// TwinCAT 3 PLC project PLC_PML
// ProgramVersion: 3.1.4023.0
// libraries:
//   PML_Base_Library, * (SPT)
//   Tc2_Math, * (Beckhoff Automation GmbH)
//   Tc2_MC2, * (Beckhoff Automation GmbH)
//   Tc2_MC2_Drive, * (Beckhoff Automation GmbH)
//   Tc2_Standard, * (Beckhoff Automation GmbH)
//   Tc2_System, * (Beckhoff Automation GmbH)
//   Tc2_Utilities, * (Beckhoff Automation GmbH)
//   Tc3_EventLogger, * (Beckhoff Automation GmbH)
//   Tc3_Module, * (Beckhoff Automation GmbH)
//   Tc3_PackML_V2, * (Beckhoff Automation GmbH)
// project tree:
//   Application/01_Application_Level_Items/02_DUT/01_ENUM/ E_PMLUnitMode.TcDUT (not stored)
//   Application/01_Application_Level_Items/02_DUT/02_STRUCT/ ST_ProductionData_HMI.TcDUT
//   Application/01_Application_Level_Items/02_DUT/03_ALIAS/ T_PackMLTags.TcDUT (not stored)
//   Application/01_Application_Level_Items/03_ITFs/ ITF_ProductionData.TcIO
//   Application/01_Application_Level_Items/04_HMI_Connections/ FB_MainModule_HMI_Connection.TcPOU (not stored), ST_PMLControl.TcDUT, ST_PMLControl_Simplified.TcDUT
//   Application/01_Application_Level_Items/999_VISU/ V_Application.TcVIS (not stored)
//   Application/01_Application_Level_Items/99_Templates/ FB_Module_TEMPLATE.TcPOU
//   Application/01_Application_Level_Items/ FB_ProductionMonitor.TcPOU
//   Application/02_MachineModules/ FB_TestMachine.TcPOU (not stored)
//   Application/03_EquipmentModules/ FB_TestEquipment.TcPOU (not stored)
//   Application/04_Components/01_Cylinder_Example/ FB_CylinderBase.TcPOU (not stored), ITF_CylinderBase.TcIO (not stored), ST_CylinderBase_HMI.TcDUT (not stored)
//   Application/ MAIN.TcPOU (not stored)
//   / GlobalTextList.TcGTLO (not stored), PlcTask.TcTTO (not stored), Visualization Manager.TcVMO (not stored)
// real-time tasks:
//   TASK PlcTask: cycle T#1ms, priority 20, ADS port 350
//   TASK VISU_TASK: cycle T#200000us, priority 30, ADS port 351
//   TASK Job Task: cycle default, priority 32
//   TASK MC-Task (MET): cycle T#2ms, priority 3, ADS port 521
//   TASK MC-Task (MPT): cycle T#10ms, priority 8, ADS port 531
// motion (NC):
//   TASK NC-Task 1 SAF: cycle T#2ms, priority 4, ADS port 501
//   TASK NC-Task 1 SVB: cycle T#10ms, priority 9, ADS port 511
//   AXIS Axis 1 (id 1)
//     General: UnitFlags=#x00000004
//     Dynamic: AccelerationMaximum=10000, DecelerationMaximum=10000, Acceleration=1000, Deceleration=1000, Jerk=1750
//     Velo: Maximum=1500
//     OtherSettings: AllowMotionCmdToSlave=true
//     encoder EncType=1
//       EncPara: ModuloFactor=720
//     drive DrvType=5
//       Analog: TorqueSetpointScale=10, ScaleFactorActTorque=0.1
//       TimeComp: TaskDelayCycles=1
//     controller CtrType=1
//       CtrPara: PriorControlFactor=1
//         Observer: BandWidth=20
//   AXIS Axis 2 (id 2)
//     General: UnitFlags=#x00000004
//     OtherSettings: AllowMotionCmdToSlave=true
//     encoder EncType=1
//     drive DrvType=5
//       Analog: TorqueSetpointScale=10, ScaleFactorActTorque=0.1
//       TimeComp: TaskDelayCycles=1
//     controller CtrType=1
//       CtrPara: PriorControlFactor=1
//         Observer: BandWidth=20

// ---- Application/01_Application_Level_Items/02_DUT/02_STRUCT/ST_ProductionData_HMI.TcDUT
TYPE ST_ProductionData_HMI :
    STRUCT
        bHMIControlAvailable    : BOOL; //Set TRUE *FROM PLC* when HMI requests can be processed
        bIncomingHMIRequest     : BOOL; //Pulses TRUE when an HMI request is issued
        bHMICommandConfirmation : BOOL; //Confirms receipt and subsequent processing of the command sent by the HMI

        bShiftLengthHMISetRequest : BOOL;
        tShiftLengthHMISetValue   : TIME;

        bShiftProductionTargetHMISetRequest : BOOL;
        nShiftProductionTargetHMISetValue   : DINT;

        bWarningMarginHMISetRequest : BOOL;
        fWarningMarginHMISetValue   : LREAL;

        bProductionRateHMISetRequest : BOOL;
        fProductionRateHMISetValue   : LREAL;

        tShiftLength           : TIME; //Specify the time duration of a shift
        nShiftProductionTarget : DINT; //Specify the desired production count by end of shift

        nCurrentAcceptableProductionCount : DINT;
        nCurrentWarningProductionCount    : DINT;
        nCurrentShiftProductionCount      : DINT; //Number of products completed so far on the current shift
        nCurrentShiftTarget               : DINT; //Expected number of completed products at the current time in the shift
        tCurrentShiftTime                 : TIME; //Time elapsed since the start of the shift
        tRemainingShiftTime               : TIME; //Time remaining in the current shift
        tShiftStartTimeStamp              : TIMESTRUCT;
        tShiftStartTimeStamp_UTC          : STRING;
        fProductionRate_Setpoint          : LREAL;
        fProductionRate_Actual            : LREAL;
        fProductionRate_Required          : LREAL;

    END_STRUCT
END_TYPE

// ---- Application/01_Application_Level_Items/04_HMI_Connections/ST_PMLControl.TcDUT
TYPE ST_PMLControl :
    STRUCT
        bNewCommand   : BOOL;
        bConfirmation : BOOL;

        eMode        : E_PMLUnitMode;
        eModeCommand : E_PMLUnitMode;

        eState        : E_PMLState;
        eStateCommand : E_PMLCommand;

        a_sModeNames : ARRAY[0..31] OF STRING;
    END_STRUCT
END_TYPE

// ---- Application/01_Application_Level_Items/04_HMI_Connections/ST_PMLControl_Simplified.TcDUT
TYPE ST_PMLControl_Simplified :
    STRUCT
        bConfirmation : BOOL;

        bClearEnabled : BOOL;
        bResetEnabled : BOOL;
        bStartEnabled : BOOL;
        bStopEnabled  : BOOL;

        bClearPressed : BOOL;
        bResetPressed : BOOL;
        bStartPressed : BOOL;
        bStopPressed  : BOOL;
    END_STRUCT
END_TYPE

// ---- Application/01_Application_Level_Items/03_ITFs/ITF_ProductionData.TcIO
INTERFACE ITF_ProductionData

PROPERTY CurrentShiftAcceptableProduction : DINT
GET
END_GET
SET
END_SET
END_PROPERTY

PROPERTY CurrentShiftProductionCount : DINT
GET
END_GET
END_PROPERTY

PROPERTY CurrentShiftTarget : DINT
GET
END_GET
END_PROPERTY

PROPERTY CurrentShiftTime : TIME
GET
END_GET
END_PROPERTY

PROPERTY CurrentShiftWarningProduction : DINT
GET
END_GET
SET
END_SET
END_PROPERTY

PROPERTY NewProductionRate : bool
GET
END_GET
END_PROPERTY

PROPERTY ProductComplete : bool
GET
END_GET
SET
END_SET
END_PROPERTY

PROPERTY ProductionRate_Actual : lreal
GET
END_GET
END_PROPERTY

PROPERTY ProductionRate_Required : lreal
GET
END_GET
SET
END_SET
END_PROPERTY

PROPERTY ProductionRate_Setpoint : lreal
GET
END_GET
SET
END_SET
END_PROPERTY

PROPERTY RateAveragingCount : DINT
GET
END_GET
SET
END_SET
END_PROPERTY

PROPERTY RemainingShiftTime : TIME
GET
END_GET
SET
END_SET
END_PROPERTY

PROPERTY ShiftComplete : BOOL
GET
END_GET
END_PROPERTY

PROPERTY ShiftLength : TIME
GET
END_GET
SET
END_SET
END_PROPERTY

PROPERTY ShiftProductionTarget : DINT
GET
END_GET
SET
END_SET
END_PROPERTY

PROPERTY WarningMargin : LREAL //0 to 100, interpreted as a percentage difference between the current rate and the required rate to meet the production target, decimal values permitted
GET
END_GET
SET
END_SET
END_PROPERTY

END_INTERFACE

// ---- Application/01_Application_Level_Items/99_Templates/FB_Module_TEMPLATE.TcPOU
FUNCTION_BLOCK FB_Module_TEMPLATE EXTENDS FB_PMLModuleBase
VAR
    //Define the Sub modules here for this module. (If any)  Also set the Interfaces in the initialize method.
    (*fbSubModule1				: FB_ApplicationModule_TEMPLATE := (ModuleName :=  'Test Module 1');
	*)
    (*fbSubModule2				: FB_ApplicationModule_TEMPLATE := (ModuleName :=  'Test Module 2');
	*)
    //temporary array of module base interfaces to be copied over to the base class a_itfPackMLBase variable
    a_ITF_PackMLBase_init : ARRAY[1..MAX_NO_OF_SUBMODULES] OF ITF_PMLModuleBase
        := [ (*	fbSubModule1,
																							 	fbSubModule2*) ];

    //Define the components here for this module. (If any) Also set the Interfaces in the initialize method.
    (*fbComponent1				: FB_ComponentBase (Extension):= (Name := 'Test Component 1');
	*)
    (*fbComponent2				: FB_ComponentBase (Extension):= (Name := 'Test Component 2');
	*)
    //temporary array of module base interfaces to be copied over to the base class a_itfPackMLBase variable
    a_ITF_Components_init : ARRAY[1..GVL_PML_Base.MAX_NO_OF_COMPONENTS] OF ITF_ComponentBase := [ (*	fbComponent1,
																											fbComponent2*)
    ];

END_VAR

//*********************************************************
//Body of block is not called by base code, only implement application
//code in CyclicUpdate or in methods called by it or its subcalls
//*********************************************************

METHOD Aborted
CASE eMode OF
    //	====================================================================PRODUCTION MODE=========================================================	
    E_PMLUnitMode.ePMLUnitMode_Production:
        ;
    //	====================================================================MANUAL MODE=============================================================	
    E_PMLUnitMode.ePMLUnitMode_Manual:
        ;
    //	=====================================================================MAINTENANCE MODE=======================================================	
    E_PMLUnitMode.ePMLUnitMode_Maintenance:
        ;
    //	=====================================================================CUSTOM MODE 1==========================================================	
    (*	E_PMLUnitMode.ePMLUnitMode_YOURCUSTOMMODE		
		;*)
    //	======================================================================INVALID MODE==========================================================	
    E_PMLUnitMode.ePMLUnitMode_Invalid:
        ;
END_CASE
END_METHOD

METHOD Aborting
//bNoStateTasksToComplete := TRUE;		// Change to False if not used

//Implement state Tasks here
(*
IF (insert your completion conditions) THEN

bStateTasksComplete := TRUE;				//Once these actions are completed successfully, set bStateTasksComplete to allow the base code to advance once all children have also reached the proper state

END_IF
*)

SUPER^.Aborting();

(*	Reference State Machine for mode specific actions - Be sure to paste above the SUPER^ Call if used - Delete if not needed

CASE eMode OF
//	====================================================================PRODUCTION MODE=========================================================	
	E_PMLUnitMode.ePMLUnitMode_Production:			
		;
//	====================================================================MANUAL MODE=============================================================	
	E_PMLUnitMode.ePMLUnitMode_Manual:				
		;
//	=====================================================================MAINTENANCE MODE=======================================================	
	E_PMLUnitMode.ePMLUnitMode_Maintenance:			
		;	
//	=====================================================================CUSTOM MODE 1==========================================================	
(*	E_PMLUnitMode.ePMLUnitMode_YOURCUSTOMMODE		
		;*)
//	======================================================================INVALID MODE==========================================================	
	E_PMLUnitMode.ePMLUnitMode_Invalid:				
		;
END_CASE
*)
END_METHOD

METHOD Clearing
//bNoStateTasksToComplete := TRUE;		// Change to False if not used

//Implement state Tasks here
(*
IF (insert your completion conditions) THEN

bStateTasksComplete := TRUE;				//Once these actions are completed successfully, set bStateTasksComplete to allow the base code to advance once all children have also reached the proper state

END_IF
*)

SUPER^.Clearing();
(*	Reference State Machine for mode specific actions - Be sure to paste above the SUPER^ Call if used - Delete if not needed

CASE eMode OF
//	====================================================================PRODUCTION MODE=========================================================	
	E_PMLUnitMode.ePMLUnitMode_Production:			
		;
//	====================================================================MANUAL MODE=============================================================	
	E_PMLUnitMode.ePMLUnitMode_Manual:				
		;
//	=====================================================================MAINTENANCE MODE=======================================================	
	E_PMLUnitMode.ePMLUnitMode_Maintenance:			
		;	
//	=====================================================================CUSTOM MODE 1==========================================================	
(*	E_PMLUnitMode.ePMLUnitMode_YOURCUSTOMMODE		
		;*)
//	======================================================================INVALID MODE==========================================================	
	E_PMLUnitMode.ePMLUnitMode_Invalid:				
		;
END_CASE
*)
END_METHOD

METHOD Complete
CASE eMode OF
    //	====================================================================PRODUCTION MODE=========================================================	
    E_PMLUnitMode.ePMLUnitMode_Production:
        ;
    //	====================================================================MANUAL MODE=============================================================	
    E_PMLUnitMode.ePMLUnitMode_Manual:
        ;
    //	=====================================================================MAINTENANCE MODE=======================================================	
    E_PMLUnitMode.ePMLUnitMode_Maintenance:
        ;
    //	=====================================================================CUSTOM MODE 1==========================================================	
    (*	E_PMLUnitMode.ePMLUnitMode_YOURCUSTOMMODE		
		;*)
    //	======================================================================INVALID MODE==========================================================	
    E_PMLUnitMode.ePMLUnitMode_Invalid:
        ;
END_CASE
END_METHOD

METHOD Completing
//bNoStateTasksToComplete := TRUE;		// Change to False if not used

//Implement state Tasks here
(*
IF (insert your completion conditions) THEN

bStateTasksComplete := TRUE;				//Once these actions are completed successfully, set bStateTasksComplete to allow the base code to advance once all children have also reached the proper state

END_IF
*)

SUPER^.Completing();

(*	Reference State Machine for mode specific actions - Be sure to paste above the SUPER^ Call if used - Delete if not needed

CASE eMode OF
//	====================================================================PRODUCTION MODE=========================================================	
	E_PMLUnitMode.ePMLUnitMode_Production:			
		;
//	====================================================================MANUAL MODE=============================================================	
	E_PMLUnitMode.ePMLUnitMode_Manual:				
		;
//	=====================================================================MAINTENANCE MODE=======================================================	
	E_PMLUnitMode.ePMLUnitMode_Maintenance:			
		;	
//	=====================================================================CUSTOM MODE 1==========================================================	
(*	E_PMLUnitMode.ePMLUnitMode_YOURCUSTOMMODE		
		;*)
//	======================================================================INVALID MODE==========================================================	
	E_PMLUnitMode.ePMLUnitMode_Invalid:				
		;
END_CASE
*)
END_METHOD

// 
// Cyclic Code
METHOD CyclicLogic
VAR
    i : UDINT; //Generic iteration value
END_VAR
// Main loop of the parent module
SUPER^.CyclicLogic();
END_METHOD

METHOD Execute
CASE eMode OF
    //	====================================================================PRODUCTION MODE=========================================================	
    E_PMLUnitMode.ePMLUnitMode_Production:
        ;
    //	====================================================================MANUAL MODE=============================================================	
    E_PMLUnitMode.ePMLUnitMode_Manual:
        ;
    //	=====================================================================MAINTENANCE MODE=======================================================	
    E_PMLUnitMode.ePMLUnitMode_Maintenance:
        ;
    //	=====================================================================CUSTOM MODE 1==========================================================	
    (*	E_PMLUnitMode.ePMLUnitMode_YOURCUSTOMMODE		
		;*)
    //	======================================================================INVALID MODE==========================================================	
    E_PMLUnitMode.ePMLUnitMode_Invalid:
        ;
END_CASE
END_METHOD

METHOD Held
CASE eMode OF
    //	====================================================================PRODUCTION MODE=========================================================	
    E_PMLUnitMode.ePMLUnitMode_Production:
        ;
    //	====================================================================MANUAL MODE=============================================================	
    E_PMLUnitMode.ePMLUnitMode_Manual:
        ;
    //	=====================================================================MAINTENANCE MODE=======================================================	
    E_PMLUnitMode.ePMLUnitMode_Maintenance:
        ;
    //	=====================================================================CUSTOM MODE 1==========================================================	
    (*	E_PMLUnitMode.ePMLUnitMode_YOURCUSTOMMODE		
		;*)
    //	======================================================================INVALID MODE==========================================================	
    E_PMLUnitMode.ePMLUnitMode_Invalid:
        ;
END_CASE
END_METHOD

METHOD Holding
//bNoStateTasksToComplete := TRUE;		// Change to False if not used

//Implement state Tasks here
(*
IF (insert your completion conditions) THEN

bStateTasksComplete := TRUE;				//Once these actions are completed successfully, set bStateTasksComplete to allow the base code to advance once all children have also reached the proper state

END_IF
*)

SUPER^.Holding();

(*	Reference State Machine for mode specific actions - Be sure to paste above the SUPER^ Call if used - Delete if not needed

CASE eMode OF
//	====================================================================PRODUCTION MODE=========================================================	
	E_PMLUnitMode.ePMLUnitMode_Production:			
		;
//	====================================================================MANUAL MODE=============================================================	
	E_PMLUnitMode.ePMLUnitMode_Manual:				
		;
//	=====================================================================MAINTENANCE MODE=======================================================	
	E_PMLUnitMode.ePMLUnitMode_Maintenance:			
		;	
//	=====================================================================CUSTOM MODE 1==========================================================	
(*	E_PMLUnitMode.ePMLUnitMode_YOURCUSTOMMODE		
		;*)
//	======================================================================INVALID MODE==========================================================	
	E_PMLUnitMode.ePMLUnitMode_Invalid:				
		;
END_CASE
*)
END_METHOD

METHOD Idle
CASE eMode OF
    //	====================================================================PRODUCTION MODE=========================================================	
    E_PMLUnitMode.ePMLUnitMode_Production:
        ;
    //	====================================================================MANUAL MODE=============================================================	
    E_PMLUnitMode.ePMLUnitMode_Manual:
        ;
    //	=====================================================================MAINTENANCE MODE=======================================================	
    E_PMLUnitMode.ePMLUnitMode_Maintenance:
        ;
    //	=====================================================================CUSTOM MODE 1==========================================================	
    (*	E_PMLUnitMode.ePMLUnitMode_YOURCUSTOMMODE		
		;*)
    //	======================================================================INVALID MODE==========================================================	
    E_PMLUnitMode.ePMLUnitMode_Invalid:
        ;
END_CASE
END_METHOD

METHOD Initialize
VAR
    i : UDINT; //Generic iteration value
END_VAR
// Define the interfaces to the different subunits (Must take place before SUPER^.initialize call)
FOR i := 1 TO MAX_NO_OF_SUBMODULES DO
    a_ITF_PackMLBase[i] := a_ITF_PackMLBase_init[i];
END_FOR

FOR i := 1 TO MAX_NO_OF_COMPONENTS DO
    a_ITF_Components[i] := a_ITF_Components_init[i];
END_FOR

// Init of the parent class object (Must be called AFTER most local init code, since the sub module interface array assignments should be made here, and then operated on within the module base init
SUPER^.Initialize();
END_METHOD

METHOD Resetting
//bNoStateTasksToComplete := TRUE;		// Change to False if not used

//Implement state Tasks here
(*
IF (insert your completion conditions) THEN

bStateTasksComplete := TRUE;				//Once these actions are completed successfully, set bStateTasksComplete to allow the base code to advance once all children have also reached the proper state

END_IF
*)

SUPER^.Resetting();

(*	Reference State Machine for mode specific actions - Be sure to paste above the SUPER^ Call if used - Delete if not needed

CASE eMode OF
//	====================================================================PRODUCTION MODE=========================================================	
	E_PMLUnitMode.ePMLUnitMode_Production:			
		;
//	====================================================================MANUAL MODE=============================================================	
	E_PMLUnitMode.ePMLUnitMode_Manual:				
		;
//	=====================================================================MAINTENANCE MODE=======================================================	
	E_PMLUnitMode.ePMLUnitMode_Maintenance:			
		;	
//	=====================================================================CUSTOM MODE 1==========================================================	
(*	E_PMLUnitMode.ePMLUnitMode_YOURCUSTOMMODE		
		;*)
//	======================================================================INVALID MODE==========================================================	
	E_PMLUnitMode.ePMLUnitMode_Invalid:				
		;
END_CASE
*)
END_METHOD

METHOD Starting
//bNoStateTasksToComplete := TRUE;		// Change to False if not used

//Implement state Tasks here
(*
IF (insert your completion conditions) THEN

bStateTasksComplete := TRUE;				//Once these actions are completed successfully, set bStateTasksComplete to allow the base code to advance once all children have also reached the proper state

END_IF
*)

SUPER^.Starting();

(*	Reference State Machine for mode specific actions - Be sure to paste above the SUPER^ Call if used - Delete if not needed

CASE eMode OF
//	====================================================================PRODUCTION MODE=========================================================	
	E_PMLUnitMode.ePMLUnitMode_Production:			
		;
//	====================================================================MANUAL MODE=============================================================	
	E_PMLUnitMode.ePMLUnitMode_Manual:				
		;
//	=====================================================================MAINTENANCE MODE=======================================================	
	E_PMLUnitMode.ePMLUnitMode_Maintenance:			
		;	
//	=====================================================================CUSTOM MODE 1==========================================================	
(*	E_PMLUnitMode.ePMLUnitMode_YOURCUSTOMMODE		
		;*)
//	======================================================================INVALID MODE==========================================================	
	E_PMLUnitMode.ePMLUnitMode_Invalid:				
		;
END_CASE
*)
END_METHOD

METHOD Stopped
CASE eMode OF
    //	====================================================================PRODUCTION MODE=========================================================	
    E_PMLUnitMode.ePMLUnitMode_Production:
        ;
    //	====================================================================MANUAL MODE=============================================================	
    E_PMLUnitMode.ePMLUnitMode_Manual:
        ;
    //	=====================================================================MAINTENANCE MODE=======================================================	
    E_PMLUnitMode.ePMLUnitMode_Maintenance:
        ;
    //	=====================================================================CUSTOM MODE 1==========================================================	
    (*	E_PMLUnitMode.ePMLUnitMode_YOURCUSTOMMODE		
		;*)
    //	======================================================================INVALID MODE==========================================================	
    E_PMLUnitMode.ePMLUnitMode_Invalid:
        ;
END_CASE
END_METHOD

METHOD Stopping
//bNoStateTasksToComplete := TRUE;		// Change to False if not used

//Implement state Tasks here
(*
IF (insert your completion conditions) THEN

bStateTasksComplete := TRUE;				//Once these actions are completed successfully, set bStateTasksComplete to allow the base code to advance once all children have also reached the proper state

END_IF
*)

SUPER^.Stopping();

(*	Reference State Machine for mode specific actions - Be sure to paste above the SUPER^ Call if used - Delete if not needed

CASE eMode OF
//	====================================================================PRODUCTION MODE=========================================================	
	E_PMLUnitMode.ePMLUnitMode_Production:			
		;
//	====================================================================MANUAL MODE=============================================================	
	E_PMLUnitMode.ePMLUnitMode_Manual:				
		;
//	=====================================================================MAINTENANCE MODE=======================================================	
	E_PMLUnitMode.ePMLUnitMode_Maintenance:			
		;	
//	=====================================================================CUSTOM MODE 1==========================================================	
(*	E_PMLUnitMode.ePMLUnitMode_YOURCUSTOMMODE		
		;*)
//	======================================================================INVALID MODE==========================================================	
	E_PMLUnitMode.ePMLUnitMode_Invalid:				
		;
END_CASE
*)
END_METHOD

METHOD Suspended
CASE eMode OF
    //	====================================================================PRODUCTION MODE=========================================================	
    E_PMLUnitMode.ePMLUnitMode_Production:
        ;
    //	====================================================================MANUAL MODE=============================================================	
    E_PMLUnitMode.ePMLUnitMode_Manual:
        ;
    //	=====================================================================MAINTENANCE MODE=======================================================	
    E_PMLUnitMode.ePMLUnitMode_Maintenance:
        ;
    //	=====================================================================CUSTOM MODE 1==========================================================	
    (*	E_PMLUnitMode.ePMLUnitMode_YOURCUSTOMMODE		
		;*)
    //	======================================================================INVALID MODE==========================================================	
    E_PMLUnitMode.ePMLUnitMode_Invalid:
        ;
END_CASE
END_METHOD

METHOD Suspending
//bNoStateTasksToComplete := TRUE;		// Change to False if not used

//Implement state Tasks here
(*
IF (insert your completion conditions) THEN

bStateTasksComplete := TRUE;				//Once these actions are completed successfully, set bStateTasksComplete to allow the base code to advance once all children have also reached the proper state

END_IF
*)

SUPER^.Suspending();

(*	Reference State Machine for mode specific actions - Be sure to paste above the SUPER^ Call if used - Delete if not needed

CASE eMode OF
//	====================================================================PRODUCTION MODE=========================================================	
	E_PMLUnitMode.ePMLUnitMode_Production:			
		;
//	====================================================================MANUAL MODE=============================================================	
	E_PMLUnitMode.ePMLUnitMode_Manual:				
		;
//	=====================================================================MAINTENANCE MODE=======================================================	
	E_PMLUnitMode.ePMLUnitMode_Maintenance:			
		;	
//	=====================================================================CUSTOM MODE 1==========================================================	
(*	E_PMLUnitMode.ePMLUnitMode_YOURCUSTOMMODE		
		;*)
//	======================================================================INVALID MODE==========================================================	
	E_PMLUnitMode.ePMLUnitMode_Invalid:				
		;
END_CASE
*)
END_METHOD

METHOD Undefined
CASE eMode OF
    //	====================================================================PRODUCTION MODE=========================================================	
    E_PMLUnitMode.ePMLUnitMode_Production:
        ;
    //	====================================================================MANUAL MODE=============================================================	
    E_PMLUnitMode.ePMLUnitMode_Manual:
        ;
    //	=====================================================================MAINTENANCE MODE=======================================================	
    E_PMLUnitMode.ePMLUnitMode_Maintenance:
        ;
    //	=====================================================================CUSTOM MODE 1==========================================================	
    (*	E_PMLUnitMode.ePMLUnitMode_YOURCUSTOMMODE		
		;*)
    //	======================================================================INVALID MODE==========================================================	
    E_PMLUnitMode.ePMLUnitMode_Invalid:
        ;
END_CASE
END_METHOD

METHOD Unholding
//bNoStateTasksToComplete := TRUE;		// Change to False if not used

//Implement state Tasks here
(*
IF (insert your completion conditions) THEN

bStateTasksComplete := TRUE;				//Once these actions are completed successfully, set bStateTasksComplete to allow the base code to advance once all children have also reached the proper state

END_IF
*)

SUPER^.Unholding();

(*	Reference State Machine for mode specific actions - Be sure to paste above the SUPER^ Call if used - Delete if not needed

CASE eMode OF
//	====================================================================PRODUCTION MODE=========================================================	
	E_PMLUnitMode.ePMLUnitMode_Production:			
		;
//	====================================================================MANUAL MODE=============================================================	
	E_PMLUnitMode.ePMLUnitMode_Manual:				
		;
//	=====================================================================MAINTENANCE MODE=======================================================	
	E_PMLUnitMode.ePMLUnitMode_Maintenance:			
		;	
//	=====================================================================CUSTOM MODE 1==========================================================	
(*	E_PMLUnitMode.ePMLUnitMode_YOURCUSTOMMODE		
		;*)
//	======================================================================INVALID MODE==========================================================	
	E_PMLUnitMode.ePMLUnitMode_Invalid:				
		;
END_CASE
*)
END_METHOD

METHOD Unsuspending
//bNoStateTasksToComplete := TRUE;		// Change to False if not used

//Implement state Tasks here
(*
IF (insert your completion conditions) THEN

bStateTasksComplete := TRUE;				//Once these actions are completed successfully, set bStateTasksComplete to allow the base code to advance once all children have also reached the proper state

END_IF
*)

SUPER^.Unsuspending();

(*	Reference State Machine for mode specific actions - Be sure to paste above the SUPER^ Call if used - Delete if not needed

CASE eMode OF
//	====================================================================PRODUCTION MODE=========================================================	
	E_PMLUnitMode.ePMLUnitMode_Production:			
		;
//	====================================================================MANUAL MODE=============================================================	
	E_PMLUnitMode.ePMLUnitMode_Manual:				
		;
//	=====================================================================MAINTENANCE MODE=======================================================	
	E_PMLUnitMode.ePMLUnitMode_Maintenance:			
		;	
//	=====================================================================CUSTOM MODE 1==========================================================	
(*	E_PMLUnitMode.ePMLUnitMode_YOURCUSTOMMODE		
		;*)
//	======================================================================INVALID MODE==========================================================	
	E_PMLUnitMode.ePMLUnitMode_Invalid:				
		;
END_CASE
*)
END_METHOD

END_FUNCTION_BLOCK

// ---- Application/01_Application_Level_Items/FB_ProductionMonitor.TcPOU
FUNCTION_BLOCK FB_ProductionMonitor IMPLEMENTS ITF_ProductionData
VAR CONSTANT
    //Constant declarations
    PRODUCTION_DATA_ALARM_COUNT : UDINT := 16;
END_VAR
VAR PERSISTENT
    //ITF_ProductionData internal variables
    tShiftLength             : TIME  := T#10M;
    nShiftProductionTarget   : DINT  := 1000;
    fWarningMargin           : LREAL := 10;
    fProductionRate_Setpoint : LREAL := 30;
    nRateAveragingCount      : DINT  := 10;
END_VAR
VAR
    //ITF_ProductionData internal variables + Other Production related variables
    bShiftComplete                    : BOOL;
    bProductComplete                  : BOOL;
    nCurrentShiftProductionCount      : INT;
    nCurrentShiftTarget               : DINT;
    tCurrentShiftTime                 : TIME;
    tRemainingShiftTime               : TIME;
    nCurrentWarningProductionCount    : DINT;
    nCurrentAcceptableProductionCount : DINT;

    fProductionRate_Required : LREAL;
    fProductionRate_Actual   : LREAL;

    a_nLastProductTimestamps  : ARRAY[1..100] OF ULINT; //Array of ULINT values (1 unit = 1ns) for the relative time of each of the last 100 completed products
    fbShiftTimer              : TON;
    fbProductComplete_RT      : R_TRIG;
    bNewProductionRate        : BOOL;
    fLastTargetProductionRate : LREAL;

    bResetMaxProductionCount   : BOOL;
    bResetTotalProductionCount : BOOL;

    nMaxProductionCount   : DINT;
    nTotalProductionCount : DINT;

    stProductionDataHMI          : ST_ProductionData_HMI;
    fbFIFO                       : FB_FIFO_ULINT_Array;
    a_fbProductionDataAlarms     : ARRAY[1..PRODUCTION_DATA_ALARM_COUNT] OF FB_TcAlarm;
    fTemp                        : LREAL;
    bInitialized                 : BOOL;
    initialize                   : INT;
    fLastProductionRate_Setpoint : LREAL;
END_VAR

PROPERTY CurrentShiftAcceptableProduction : DINT
GET
END_GET
SET
END_SET
END_PROPERTY

PROPERTY CurrentShiftProductionCount : DINT
GET
CurrentShiftProductionCount := nCurrentShiftProductionCount;
END_GET
END_PROPERTY

PROPERTY CurrentShiftTarget : DINT
GET
CurrentShiftTarget := nCurrentShiftTarget;
END_GET
END_PROPERTY

PROPERTY CurrentShiftTime : TIME
GET
CurrentShiftTime := tCurrentShiftTime;
END_GET
END_PROPERTY

PROPERTY CurrentShiftWarningProduction : DINT
GET
END_GET
SET
END_SET
END_PROPERTY

METHOD HMICommunication : BOOL
VAR_INPUT
END_VAR
//Production Data================================================================================================================================================

//Process HMI requests
IF stProductionDataHMI.bIncomingHMIRequest AND NOT stProductionDataHMI.bHMICommandConfirmation
    THEN //If a request has been issued by the HMI, and a previous request has not just E_SequenceState.Finished being processed
    IF stProductionDataHMI.bShiftProductionTargetHMISetRequest THEN
        nShiftProductionTarget                      := stProductionDataHMI.nShiftProductionTargetHMISetValue;
        stProductionDataHMI.bHMICommandConfirmation := TRUE; //Confirm that the request has been processed
    END_IF

    IF stProductionDataHMI.bWarningMarginHMISetRequest THEN
        fWarningMargin                              := stProductionDataHMI.fWarningMarginHMISetValue;
        stProductionDataHMI.bHMICommandConfirmation := TRUE; //Confirm that the request has been processed
    END_IF

    IF stProductionDataHMI.bShiftLengthHMISetRequest THEN
        tShiftLength                                := stProductionDataHMI.tShiftLengthHMISetValue;
        stProductionDataHMI.bHMICommandConfirmation := TRUE; //Confirm that the request has been processed
    END_IF

    IF stProductionDataHMI.bProductionRateHMISetRequest THEN
        fProductionRate_Setpoint                    := stProductionDataHMI.fProductionRateHMISetValue;
        stProductionDataHMI.bHMICommandConfirmation := TRUE; //Confirm that the request has been processed
    END_IF
END_IF

//Update HMI Status Info
stProductionDataHMI.tShiftLength                      := tShiftLength;
stProductionDataHMI.nShiftProductionTarget            := nShiftProductionTarget;
stProductionDataHMI.nCurrentShiftProductionCount      := nCurrentShiftProductionCount;
stProductionDataHMI.nCurrentShiftTarget               := nCurrentShiftTarget;
stProductionDataHMI.nCurrentAcceptableProductionCount := nCurrentAcceptableProductionCount;
stProductionDataHMI.nCurrentWarningProductionCount    := nCurrentWarningProductionCount;
stProductionDataHMI.tCurrentShiftTime                 := tCurrentShiftTime;
stProductionDataHMI.tRemainingShiftTime               := tRemainingShiftTime;
stProductionDataHMI.fProductionRate_Setpoint          := F_LREAL_RoundToPlace(fProductionRate_Setpoint, 1);
stProductionDataHMI.fProductionRate_Actual            := F_LREAL_RoundToPlace(fProductionRate_Actual, 1);
stProductionDataHMI.fProductionRate_Required          := F_LREAL_RoundToPlace(fProductionRate_Required, 1);
END_METHOD

METHOD initialize : BOOL
VAR_INPUT
END_VAR
END_METHOD

METHOD Monitor : BOOL
VAR_INPUT
END_VAR
IF NOT bInitialized THEN
    initialize();
    bInitialized := TRUE;
END_IF

fbFIFO(a_FIFO := a_nLastProductTimestamps);

fbShiftTimer(IN := NOT bShiftComplete, PT := tShiftLength, Q => bShiftComplete, ET => tCurrentShiftTime);
tRemainingShiftTime := tShiftLength - tCurrentShiftTime;

IF TIME_TO_DINT(tRemainingShiftTime) > 0 THEN
    fProductionRate_Required :=
        DINT_TO_LREAL(nShiftProductionTarget - nCurrentShiftProductionCount) / (TIME_TO_LREAL(tRemainingShiftTime) / 1000 / 60);

    nCurrentAcceptableProductionCount := nCurrentShiftTarget;

    nCurrentWarningProductionCount :=
        nShiftProductionTarget
            - (LREAL_TO_DINT((fProductionRate_Actual * (1 + fWarningMargin / 100)) * (TIME_TO_LREAL(tRemainingShiftTime) / 1000 / 60)));

    IF nCurrentWarningProductionCount < 0 THEN
        nCurrentWarningProductionCount := 0;
    END_IF
END_IF

fbProductComplete_RT(CLK := bProductComplete);

IF fbProductComplete_RT.Q THEN
    nCurrentShiftProductionCount := nCurrentShiftProductionCount + 1;
    nTotalProductionCount        := nTotalProductionCount + 1;

    IF nCurrentShiftProductionCount > nMaxProductionCount THEN
        nMaxProductionCount := nCurrentShiftProductionCount;
    END_IF

    fbFIFO.AddEntry(nEntry := F_GetSystemTime());
END_IF

IF (fbFIFO.EntryCount > nRateAveragingCount) THEN
    fbFIFO.RemoveEntry();
END_IF

fTemp := (TIME_TO_LREAL(ULINT_TO_TIME(fbFIFO.LastInValue - fbFIFO.NextOutValue)) / 10000 / 1000 / 60);

IF fTemp > 0 AND fbFIFO.EntryCount > 1 THEN
    fProductionRate_Actual := F_LREAL_RoundToPlace(DINT_TO_LREAL(fbFIFO.EntryCount - 1) / fTemp, 2);
END_IF

IF TIME_TO_DINT(tShiftLength) > 0 THEN
    nCurrentShiftTarget := LREAL_TO_DINT((TIME_TO_LREAL(tCurrentShiftTime) / TIME_TO_LREAL(tShiftLength)) * DINT_TO_LREAL(nShiftProductionTarget));
END_IF

IF bShiftComplete THEN
    nCurrentShiftProductionCount := 0;
END_IF

IF bResetMaxProductionCount THEN
    nMaxProductionCount := nCurrentShiftProductionCount;
END_IF

IF bResetTotalProductionCount THEN
    nTotalProductionCount := 0;
END_IF

IF fProductionRate_Setpoint <> fLastTargetProductionRate THEN
    bNewProductionRate := TRUE;
ELSE
    bNewProductionRate := FALSE;
END_IF

fLastTargetProductionRate := fProductionRate_Setpoint;
END_METHOD

PROPERTY NewProductionRate : BOOL
GET
NewProductionRate := bNewProductionRate;
END_GET
END_PROPERTY

PROPERTY ProductComplete : BOOL
GET
ProductComplete := bProductComplete;
END_GET
SET
bProductComplete := ProductComplete;
END_SET
END_PROPERTY

PROPERTY ProductionRate_Actual : LREAL
GET
ProductionRate_Actual := fProductionRate_Actual;
END_GET
END_PROPERTY

PROPERTY ProductionRate_Required : LREAL
GET
ProductionRate_Required := fProductionRate_Required;
END_GET
SET
fProductionRate_Required := ProductionRate_Required;
END_SET
END_PROPERTY

PROPERTY ProductionRate_Setpoint : LREAL
GET
ProductionRate_Setpoint := fProductionRate_Setpoint;
END_GET
SET
fProductionRate_Setpoint := ProductionRate_Setpoint;
END_SET
END_PROPERTY

PROPERTY RateAveragingCount : DINT
GET
RateAveragingCount := nRateAveragingCount;
END_GET
SET
nRateAveragingCount := RateAveragingCount;
END_SET
END_PROPERTY

PROPERTY RemainingShiftTime : TIME
GET
END_GET
SET
END_SET
END_PROPERTY

PROPERTY ShiftComplete : BOOL
GET
ShiftComplete := bShiftComplete;
END_GET
END_PROPERTY

PROPERTY ShiftLength : TIME
GET
ShiftLength := tShiftLength;
END_GET
SET
tShiftLength := ShiftLength;
END_SET
END_PROPERTY

PROPERTY ShiftProductionTarget : DINT
GET
ShiftProductionTarget := nShiftProductionTarget;
END_GET
SET
nShiftProductionTarget := ShiftProductionTarget;
END_SET
END_PROPERTY

PROPERTY WarningMargin : LREAL
GET
WarningMargin := fWarningMargin;
END_GET
SET
fWarningMargin := WarningMargin;
END_SET
END_PROPERTY

END_FUNCTION_BLOCK
